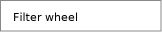
VISUALIZATION VISU_AxesConfig_FilterWheel  // 162x32
    Label (10,5 150x25), "Filter wheel"
END_VISUALIZATION

(* stored: Version 1.1.0.1, ProductVersion 3.1.4018.5
   Visu VISU_AxesConfig_FilterWheel: Id {9c37dd55-22ba-4055-b934-420b1497a856} *)
